// TIA Portal V20 export
TYPE "LWONIK_typeFromSafetyEstopStatus"
// stored: Access Published
   STRUCT
      mainOpEMO : Bool;
      processPnPEMO : Bool;
      unloadingEMO : Bool;
      weightngBoxEMO : Bool;
      hotPressEMO : Bool;
      pHmi01EMO : Bool;
      pHmi02EMO : Bool;
      pHmi01ForceDisconnected : Bool;
      pHmi02ForceDisconnected : Bool;
      ba10EMO : Bool;
      ba15EMO : Bool;
      ba30EMO : Bool;
      ba40EMO : Bool;
      ba100EMO : Bool;
      insideNoEStopPressed : Bool;
      insideEStop : Bool;
      outsideEStop : Bool;
   END_STRUCT;
END_TYPE
